// SIMATIC S7-200 project (STEP 7-Micro/WIN), CPU 224XP REL 02.01

ORGANIZATION_BLOCK MAIN:OB1
TITLE=PROGRAM COMMENTS
BEGIN
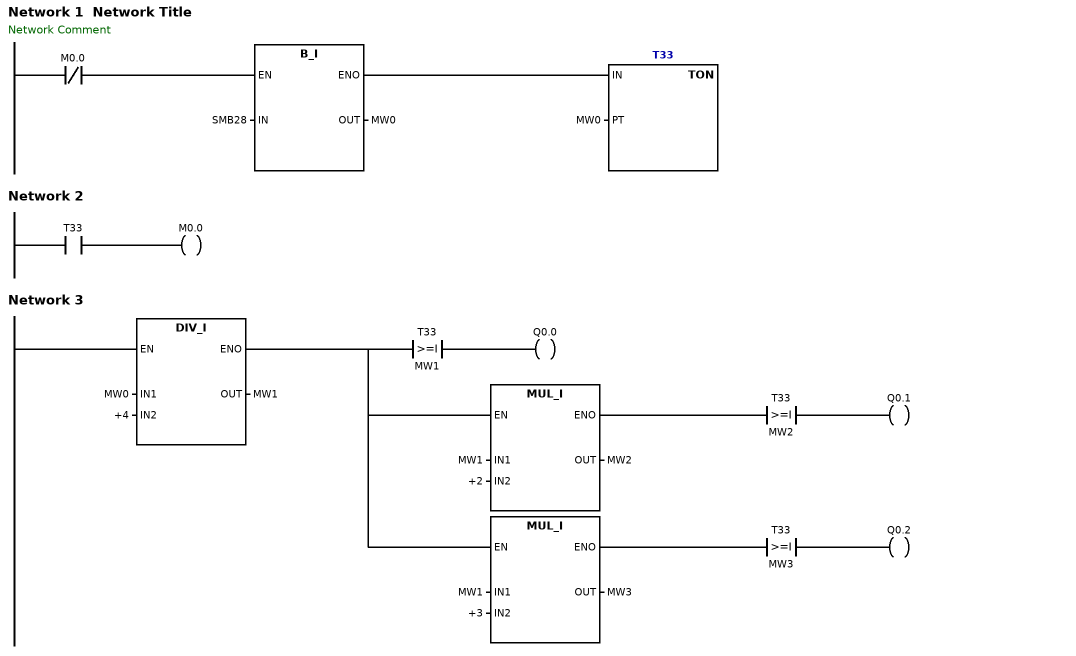
Network 1 // Network Title
// Network Comment
LDN    M0.0
BTI    SMB28, MW0
AENO
TON    T33, MW0
Network 2
LD     T33
=      M0.0
Network 3
MOVW   MW0, MW1
AENO
/I     +4, MW1
AENO
LPS
AW>=   T33, MW1
=      Q0.0
LRD
MOVW   MW1, MW2
AENO
*I     +2, MW2
AENO
AW>=   T33, MW2
=      Q0.1
LPP
MOVW   MW1, MW3
AENO
*I     +3, MW3
AENO
AW>=   T33, MW3
=      Q0.2
END_ORGANIZATION_BLOCK
